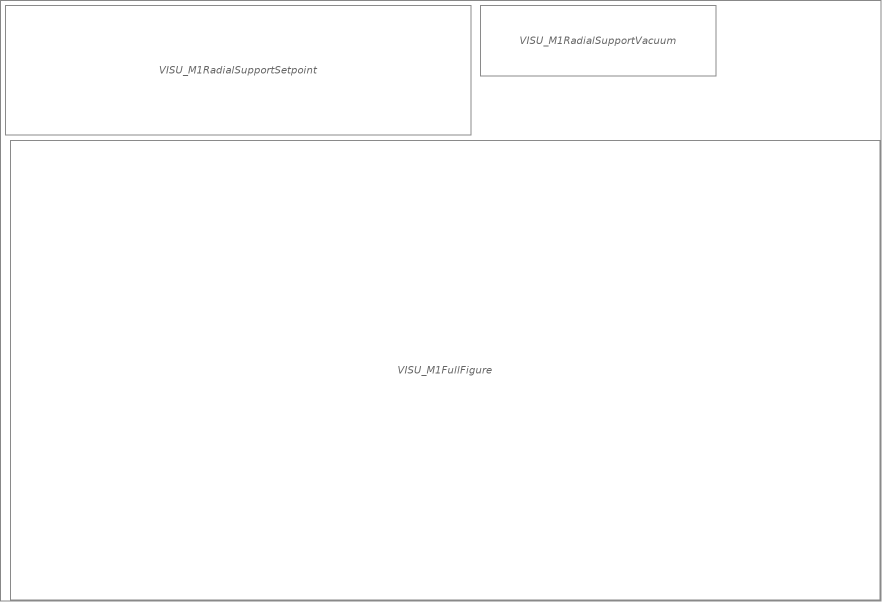
VISUALIZATION VISU_M1RadialSupport  // 882x602
VAR_IN_OUT
	ref : M1RadialSupport;
    widget : M1RadialSupportWidget;
    m1Ref : M1;
    m1Widget : M1Widget;
END_VAR
    Frame (5,5 466x130)
        shows VISU_M1RadialSupportSetpoint(ref := ref, widget := widget)
    Frame (10,140 870x460)
        shows VISU_M1FullFigure(ref := m1Ref, widget := m1Widget)
    Frame (480,5 236x71)
        shows VISU_M1RadialSupportVacuum(ref := ref, widget := widget)
END_VISUALIZATION

(* stored: Version 1.1.0.1, ProductVersion 3.1.4019.2
   Visu VISU_M1RadialSupport: Id {6a48ecc5-de6f-4438-9654-1ace94740dcf} *)
